{attribute 'enable_dynamic_creation'}
FUNCTION_BLOCK FB_Executor
VAR_INPUT
END_VAR
VAR_OUTPUT
END_VAR
VAR
	{attribute 'TcEncoding':='UTF-8'}
	_id : T_MaxString;
	_done : BOOL;
	_start : BOOL;
	_resume : BOOL;
	_passive_abort : BOOL;
	_quit : BOOL;
	_upstream_aborting : BOOL := TRUE;
	 {attribute 'TcAnalytics'}
	 _state :E_FutureExecutionState := E_FutureExecutionState.idle;
	_last_state  :E_FutureExecutionState;
	_error_id : UDINT;
	_aborting :BOOL;
	_quitting :BOOL;
	_interface_container : InterfaceContainer := 0;
	_job_event_reporters : ARRAY[1..10] OF InterfaceObserver;
	_future_creator : InterfaceTaskCreator;
	_future : InterfaceFuture;
	_parent_executor : REFERENCE TO FB_Executor REF= 0;
	_persistent_job : BOOL;
END_VAR

(*abort method

*)
METHOD abort : BOOL // Return TRUE if finish.
VAR_INPUT
END_VAR
IF _state = E_FutureExecutionState.init OR
   _state = E_FutureExecutionState.process OR
   _state = E_FutureExecutionState.quit THEN
   	_start := FALSE;
	_passive_abort := TRUE;	
	THIS^.execute();
	abort := FALSE;
ELSE
	IF _state = E_FutureExecutionState.abort THEN
		THIS^.execute();
		abort := NOT _aborting;
	ELSE
		abort := TRUE;
	END_IF
END_IF
END_METHOD

PROPERTY busy : BOOL
GET
busy := (	_state = E_FutureExecutionState.init OR	
			_state = E_FutureExecutionState.process OR 
			_state = E_FutureExecutionState.quit
		);
END_GET
END_PROPERTY

PROPERTY children : InterfaceContainer // Accesser for interface pointer to child container instance.
GET
children := _interface_container;
END_GET
END_PROPERTY

PROPERTY continuous_mode : bool // Make true if keep executing state after all jobs be finished.
SET
IF _future <> 0 THEN
	IF __QUERYINTERFACE(_future, _interface_container) THEN
		_interface_container.continuous_mode := continuous_mode;
	END_IF	
END_IF
END_SET
END_PROPERTY

METHOD create_container : InterfaceContainer // Make container object onto child.
VAR_INPUT
	container_type : ContainerType; // specify container type
	name: STRING;	// specify future name
END_VAR
VAR
	delete_existing_container : BOOL;
	created_future : InterfaceFuture;
END_VAR
IF _interface_container <> 0 THEN
 	IF _interface_container.reset(FALSE) THEN
		delete_existing_container := TRUE;
	ELSE
		delete_existing_container := FALSE;
	END_IF
ELSE
	delete_existing_container := TRUE;
END_IF

IF delete_existing_container THEN
	CASE container_type OF
		ContainerType.BATCH:
			created_future := create_future(GVL.batch_job_container_creator, name);
			created_future.executor.persistent_job := FALSE;
		ContainerType.PARALLEL:
			created_future := create_future(GVL.parallel_job_container_creator, name);
			created_future.executor.persistent_job := FALSE;
		ContainerType.QUEUE:
			created_future := create_future(GVL.queue_job_container_creator, name);
			created_future.executor.persistent_job := TRUE;
		ContainerType.PARALLEL_QUEUE:
			created_future := create_future(GVL.parallel_queue_job_container_creator, name);
			created_future.executor.persistent_job := TRUE;
	END_CASE
	THIS^.init();
	create_container := THIS^.children;
END_IF
END_METHOD

METHOD create_future : InterfaceFuture // Create future dynamically.
VAR_INPUT
	creator : InterfaceTaskCreator; // Specify creator object by which Interface Task Creator implemented.
	future_name: STRING; // Spcfigy future name.
END_VAR
_future_creator := creator;
IF _future_creator <> 0 THEN
	THIS^.future := creator.create_future(future_name);
END_IF
create_future := _future;
END_METHOD

{attribute 'OPC.UA.DA.Property' := '1'}
{attribute 'monitoring' := 'call'}
{attribute 'OPC.UA.DA.Description' := 'Current state of this executor object.'}
PROPERTY current_state : E_FutureExecutionState // Get current job state
GET
current_state := _state;
END_GET
END_PROPERTY

PROPERTY done : BOOL // Present true if process be finished.
GET
done := _done;
END_GET
END_PROPERTY

METHOD error_reset : BOOL
VAR_INPUT
END_VAR
VAR
	i_err_rst : INT;
END_VAR
IF _future <> 0 THEN
	IF _future.error_reset() THEN
		error_reset := TRUE;
		FOR i_err_rst := 1 TO 10 DO
			IF _job_event_reporters[i_err_rst] <> 0 THEN
				_job_event_reporters[i_err_rst].subscribe_job_event(
							subject := 'ERROR_RESET',
							old_state := _last_state,
							new_state := _state,
							record_time := F_GetSystemTime(),
							executor := THIS^
					);
			END_IF
		END_FOR
	ELSE
		error_reset := FALSE;
	END_IF
	_error_id := _future.nErrorID;
ELSE
	_error_id := 0;
	error_reset := TRUE;
END_IF
END_METHOD

METHOD execute : BOOL // Execute future process and return TRUE if all task are finished.
VAR_INST
	_state_mem :E_FutureExecutionState;
	_logging :BOOL;
	delay : TIME := T#3S;
	sleep : TON;
END_VAR
VAR
	_executor : REFERENCE TO FB_Executor;
	start_all_children : BOOL;
	exe: INT;
	i_check : INT;
	i_call : INT;
	bAllReportedSuccessfully : BOOL;
END_VAR
IF _future = 0 THEN
	execute := TRUE;
	RETURN;
ELSE
	execute := FALSE;
END_IF

IF _passive_abort THEN
	_state := E_FutureExecutionState.abort;
	IF _error_id = 0 THEN
		_error_id := E_ErrorId.PASSIVE_ABORT;
	END_IF
	_passive_abort := FALSE;
END_IF

IF _quit THEN
	_state := E_FutureExecutionState.quit;
END_IF
_quit := FALSE;

CASE _state OF
	E_FutureExecutionState.idle:
		ADSLOGSTR(msgCtrlMask := ADSLOG_MSGTYPE_LOG, msgFmtStr := TO_STRING(_future.state), strArg := '');
		IF _future.state = E_FutureExecutionState.idle OR 
			_future.state = E_FutureExecutionState.finish THEN
			IF init() THEN
				_state := E_FutureExecutionState.init;
			END_IF
		END_IF
	E_FutureExecutionState.init:
		IF _future.init() THEN
			IF _future.nErrorID = 0 THEN
				_state := E_FutureExecutionState.wait_for_process;
			ELSE
				_last_state := E_FutureExecutionState.init;
				_error_id := _future.nErrorID;
				_state := E_FutureExecutionState.abort;
			END_IF
		END_IF
	E_FutureExecutionState.wait_for_process: 
		IF _start THEN
			_state := E_FutureExecutionState.process;
			_start := FALSE;
		END_IF
	E_FutureExecutionState.process: 
		IF _future.execute() THEN
			IF _future.nErrorID = 0 THEN
				_state := E_FutureExecutionState.quit;
				_done := TRUE;
			ELSE
				_error_id := _future.nErrorID;
				_state := E_FutureExecutionState.abort;
			END_IF
		END_IF
	E_FutureExecutionState.abort:
		IF _aborting THEN
			_resume := FALSE;
			IF _upstream_aborting AND __ISVALIDREF(_parent_executor) THEN
				_parent_executor.abort();				
			END_IF
			IF _future.abort() THEN
				_aborting := FALSE;
			END_IF
		ELSIF _resume THEN
			_state := _last_state;
			IF _error_id = E_ErrorId.PASSIVE_ABORT THEN
				_error_id := 0;
			END_IF
			_resume := FALSE;
		END_IF
	E_FutureExecutionState.quit:
		IF _future.quit() THEN
			IF _future.nErrorID = 0 THEN
				_state := E_FutureExecutionState.finish;
			ELSE
				_error_id := _future.nErrorID;
				_state := E_FutureExecutionState.abort;
			END_IF
			_quitting := FALSE;
		END_IF
	E_FutureExecutionState.finish:
		IF NOT _logging THEN
			execute := TRUE;
		END_IF
END_CASE

IF _state <> _state_mem THEN
	_last_state := _state_mem;

	IF _state = E_FutureExecutionState.init OR
		_state = E_FutureExecutionState.process OR
		_state = E_FutureExecutionState.quit THEN
		_error_id := 0;
	END_IF

	IF _state = E_FutureExecutionState.abort THEN
		_aborting := TRUE;
	END_IF
	
	IF _state = E_FutureExecutionState.quit THEN
		sleep(IN := FALSE);
		_quitting := TRUE;
	END_IF
		
	// Check if any reporter is assigned and if the state is reportable
	IF _state >= E_FutureExecutionState.idle AND _state <= E_FutureExecutionState.finish THEN
		FOR i_check := 1 TO 10 DO
			IF _job_event_reporters[i_check] <> 0 THEN
				_logging := TRUE;
				EXIT; // Found a reporter, set logging and exit loop
			END_IF
		END_FOR
	END_IF
END_IF

_state_mem := _state;

IF _logging THEN
    bAllReportedSuccessfully := TRUE; // Initialize before the loop

    FOR i_call := 1 TO 10 DO
        IF _job_event_reporters[i_call] <> 0 THEN
            IF NOT _job_event_reporters[i_call].subscribe_job_event(
                    subject := 'TRANSITION',
                    old_state := _last_state,
                    new_state := _state,
                    record_time := F_GetSystemTime(),
                    executor := THIS^
            ) THEN
                bAllReportedSuccessfully := FALSE; // If any reporter is "busy" or fails, keep _logging for next cycle potentially
            END_IF
        END_IF
    END_FOR

    IF bAllReportedSuccessfully THEN
        _logging := FALSE; // All *active* reporters were successful
    END_IF
END_IF

IF _future <> 0 THEN
	_future.state := _state;
END_IF
END_METHOD

PROPERTY future : InterfaceFuture // Set future instance direct.
GET
future := _future;
END_GET
SET
_future := future;
_future.state := _state;
_future.executor REF= THIS^;
IF NOT __QUERYINTERFACE(_future, _interface_container) THEN
	_interface_container := 0;
END_IF
END_SET
END_PROPERTY

PROPERTY future_creator : InterfaceTaskCreator // Set creator instance.
SET
_future_creator := future_creator;
END_SET
END_PROPERTY

PROPERTY id : T_MaxString // Get job id.
GET
id := _id;
END_GET
SET
_id := id;
END_SET
END_PROPERTY

METHOD init : BOOL // Return TRUE if finish.
VAR_INPUT
END_VAR
_done := FALSE;
_passive_abort := FALSE;
_start := FALSE;
_state := E_FutureExecutionState.init;
_error_id := 0;
IF _future <> 0 THEN
	_future.init();
END_IF

INIT := TRUE;
END_METHOD

PROPERTY last_state : E_FutureExecutionState
GET
last_state := _last_state;
END_GET
END_PROPERTY

PROPERTY nErrorID : UDINT // Present error code when each process,init(), execute(), quit() are finished. '0' represent normal condition without any errors.
GET
nErrorID := _error_id;
END_GET
END_PROPERTY

PROPERTY parent_executor : REFERENCE TO FB_Executor
GET
parent_executor REF= _parent_executor;
END_GET
SET
_parent_executor REF= parent_executor;
END_SET
END_PROPERTY

PROPERTY persistent_job : BOOL
GET
persistent_job := _persistent_job;
END_GET
SET
_persistent_job := persistent_job;
END_SET
END_PROPERTY

METHOD quit : BOOL // Return TRUE if finish.
VAR_INPUT
END_VAR
IF _state = E_FutureExecutionState.init OR
   _state = E_FutureExecutionState.process OR
   _state = E_FutureExecutionState.quit THEN
	_quit := TRUE;	
END_IF

IF 	_quit AND _state = E_FutureExecutionState.quit THEN
	quit := NOT _quitting;
ELSE
	quit := TRUE;
END_IF
END_METHOD

PROPERTY ready : BOOL
GET
ready := _state = E_FutureExecutionState.wait_for_process;
END_GET
END_PROPERTY

METHOD reset : BOOL // Return TRUE if finish.
VAR_INPUT
	deep : BOOL := FALSE;
END_VAR
VAR
	_reset_children :BOOL := FALSE;
END_VAR
// Waiting finish process and remove jobs from container items.
IF THIS^.busy THEN
	THIS^.abort();
ELSIF _interface_container <> 0 AND ( NOT _persistent_job OR deep) THEN
	IF _interface_container.reset(deep) THEN
		_reset_children := TRUE;
	END_IF
ELSE
	_reset_children := TRUE;
END_IF

// Remove my future.
IF _reset_children AND _future <> 0 THEN
	IF  NOT _persistent_job OR deep THEN
		IF _future_creator <> 0 THEN
			_future := _future_creator.destroy_future(_future);
		ELSIF _future.init() THEN
			_future.state := E_FutureExecutionState.idle;
			_future := 0;
		END_IF
		IF _future = 0 THEN
			_interface_container := 0;
			reset := TRUE;
		END_IF
	ELSE
		IF _future.init() THEN
			reset := TRUE;
		END_IF
	END_IF
END_IF
END_METHOD

METHOD resume : BOOL
VAR_INST
	_executor : REFERENCE TO FB_Executor;
END_VAR
_resume := TRUE;
IF _interface_container <> 0 THEN
	IF NOT _interface_container.resume() THEN
		_resume := FALSE;
	END_IF
END_IF
IF NOT _resume THEN
	_future.execute();
END_IF
resume := _resume;
END_METHOD

METHOD start : BOOL
VAR
	_start_children :BOOL := FALSE;
END_VAR
// Send start signal to children.
IF _interface_container <> 0 THEN
	IF _interface_container.start() THEN
		_start_children := TRUE;
	END_IF
ELSE
	_start_children := TRUE;
END_IF

// Start my future.
IF _start_children THEN
	_start := _state = E_FutureExecutionState.wait_for_process;
	start := TRUE;
END_IF
END_METHOD

PROPERTY uid : T_MaxString
GET
VAR
	_eval_executor : REFERENCE TO FB_Executor;
	_uid : T_MaxString;
END_VAR
_eval_executor REF= _parent_executor;
_uid := _id;
REPEAT
	_uid := CONCAT('/',_uid);
	IF __ISVALIDREF(_eval_executor) THEN
		_uid := CONCAT(_eval_executor.id, _uid);
		_eval_executor REF= _eval_executor._parent_executor;
	END_IF
UNTIL
	NOT __ISVALIDREF(_eval_executor)
END_REPEAT

uid := _uid;
END_GET
END_PROPERTY

PROPERTY upstream_aborting : BOOL
GET
upstream_aborting := _upstream_aborting;
END_GET
SET
_upstream_aborting := upstream_aborting;
END_SET
END_PROPERTY

METHOD Subscribe : BOOL
VAR_INPUT
    observer : InterfaceObserver;
END_VAR

VAR
    i: INT;
    bSubscribed: BOOL := FALSE; // Flag to check if already subscribed
    idxEmpty: INT := 0; // Index of first empty slot
END_VAR

IF observer = 0 THEN
    Subscribe := FALSE;
    RETURN;
END_IF

// Check if already subscribed or find an empty slot
FOR i := 1 TO 10 DO // Assuming array size is 10
    IF _job_event_reporters[i] = observer THEN
        bSubscribed := TRUE;
        EXIT;
    END_IF
    IF idxEmpty = 0 AND _job_event_reporters[i] = 0 THEN
        idxEmpty := i;
    END_IF
END_FOR

IF bSubscribed THEN
    Subscribe := TRUE; // Already subscribed, consider it a success
    RETURN;
END_IF

IF idxEmpty <> 0 THEN
    _job_event_reporters[idxEmpty] := observer;
    Subscribe := TRUE;
ELSE
    Subscribe := FALSE; // Array is full
END_IF
END_METHOD

METHOD Unsubscribe : BOOL
VAR_INPUT
    observer : InterfaceObserver;
END_VAR

VAR
    i: INT;
    bFound: BOOL := FALSE;
END_VAR

IF observer = 0 THEN
    Unsubscribe := FALSE;
    RETURN;
END_IF

FOR i := 1 TO 10 DO // Assuming array size is 10
    IF _job_event_reporters[i] = observer THEN
        _job_event_reporters[i] := 0; // Remove observer
        bFound := TRUE;
        EXIT; // Exit after finding and removing
    END_IF
END_FOR

Unsubscribe := bFound;
END_METHOD

END_FUNCTION_BLOCK

(* stored: Version 1.1.0.1, ProductVersion 3.1.4024.13
   POU FB_Executor: Id {09518444-1d1d-452e-9e8f-647b2f8c5e33}, SpecialFunc None
   Method abort: Id {4a5ac73d-0cc9-4d9e-84fc-915012ed9ab4}
   Property busy: Id {4599679c-a89e-4edf-a42c-abccebfc0bd6}
   Get Get: Id {31f63b84-9fea-4918-ac72-b4f3235d586f}
   Property children: Id {db662496-7037-4faa-b7c6-23f2d18395d1}
   Get Get: Id {b5bd3ec9-ba69-4ba1-8ec7-43c8c7dc9772}
   Property continuous_mode: Id {f813b158-0532-443d-867f-f3f4c7f7b526}
   Set Set: Id {d13ba071-7139-40fe-a4d6-bf1103d7257f}
   Method create_container: Id {3ee4e0b3-d5fa-4216-b2fc-b9b451f3b414}
   Method create_future: Id {4dbfc7cf-833f-45fc-a4dd-f4a1587ef4ef}
   Property current_state: Id {9bdc45ea-e038-402f-9e8e-3b1c363b70b4}
   Get Get: Id {6d7ef6bc-7830-4957-91e4-53fd4bd8f4ba}
   Property done: Id {4120264c-9741-4f55-a3ec-37db4b2fdd1d}
   Get Get: Id {adfb9284-a38c-48f0-99cc-b8f7d36d7c03}
   Method error_reset: Id {2f58a820-9692-4e5a-84bc-d2abdb71e852}
   Method execute: Id {12a00ca6-fc73-4fe5-8b5c-2a7a9dcde6d1}
   Property future: Id {a5f34e34-fd86-442a-a2b3-dcfdacffba84}
   Get Get: Id {ea3475fd-42f3-40d5-80b9-94fefa3dce7f}
   Set Set: Id {1c600ba1-a530-4be6-883c-03a190a9123a}
   Property future_creator: Id {4ef3d23b-70fc-42e7-92d1-5df42cf5ccf9}
   Set Set: Id {73c997cd-b03a-40d8-97e1-94183b40cdc9}
   Property id: Id {cfcf1743-1715-4af2-a0a4-cd9f1ebd1808}
   Get Get: Id {5863c94c-93ce-4810-8c6f-f18910d5e32a}
   Set Set: Id {9e8cd938-613c-4a5e-bd20-a66e0b88a473}
   Method init: Id {204f5707-ec01-4438-ae9f-8cbe74e0162c}
   Property last_state: Id {02f59fbb-3554-446d-b45f-63f705bf0087}
   Get Get: Id {68fa5637-46a2-41df-8fb4-fd6bb35fe1de}
   Property nErrorID: Id {b8e1cf4d-b2aa-4996-8037-fe94c831ada6}
   Get Get: Id {279bd7d5-87e3-414a-919d-b55c6d45fe5f}
   Property parent_executor: Id {b57cb923-713c-4924-8cfc-cae55fa1c52b}
   Get Get: Id {e78d9b69-dec8-4381-b9cd-280132473f08}
   Set Set: Id {577406ef-8da9-4b14-a0b7-e722091103f8}
   Property persistent_job: Id {b89a0e73-a4d3-4c48-90ea-4677cb6b1e21}
   Get Get: Id {4e0a202e-d946-4c95-8d14-6311de03e544}
   Set Set: Id {221196e4-1427-4553-95a0-98128bf59f13}
   Method quit: Id {a3ed0ceb-2877-462b-84db-f716a8c9598e}
   Property ready: Id {a76eb28b-8e38-458e-b69a-c73f1b377610}
   Get Get: Id {b15bc61f-5bad-464a-9e63-5e877e3aa3c7}
   Method reset: Id {32d5d6a5-da71-471a-b4b9-590194585265}
   Method resume: Id {e3dc2ca8-54b7-423a-8cca-8c4b62e978bb}
   Method start: Id {fb7671b6-91ac-4f18-8e41-b81f64039055}
   Property uid: Id {564a3395-593c-4073-b553-e3a86e6b9914}
   Get Get: Id {c15a7ab7-b8a0-43cc-8050-a48bb688e753}
   Property upstream_aborting: Id {005019ae-b53c-48e8-93f8-286c00c2c383}
   Get Get: Id {63c291b8-3195-41b6-aa40-ef7a1188cf41}
   Set Set: Id {591710e5-8526-4fe9-bae8-a2b8d28c07cb}
   Method Subscribe: Id {AAAAAAAA-BBBB-CCCC-DDDD-EEEEEEEE0001}
   Method Unsubscribe: Id {AAAAAAAA-BBBB-CCCC-DDDD-EEEEEEEE0002} *)
